Fanuc KAREL source: ka00225.KL

-- PROVISIONAL review KL for V1013-1; original PC SHA256 252ef82bfacd117c2bb5dec1e0f7982433ebd5252d094ce26da0a0380edca8dd
-- Incomplete behavior may be omitted. Consult companion uncertainty JSON. Do not deploy.
PROGRAM KA00225
%NOLOCKGROUP
BEGIN
  -- UNRESOLVED_PC offsets 5-19; opcodes 22,22,1E
  -- UNRESOLVED_PC offsets 24-28; opcodes 7F
END KA00225
